{region '#Template'}
	{attribute 'Version' := '5.0.0.0'}
	{attribute 'Tags' := '"LCID": "1031", "Text": "RA, Sunprotection, Building"'}
	{attribute 'Tags' := '"LCID": "1033", "Text": "RA, Sunprotection, Building"'}
	{attribute 'Using' := '"Type": "Template", "URI": "Site"'}
	{attribute 'Using' := '"Type": "Template", "URI": "EC_ID"'}
	{attribute 'Using' := '"Type": "Template", "URI": "ST_BA_Sunblind"'}
	{attribute 'Description' := '"LCID": "1031", "Text": "Sonnenschutz Vereisungsschutz"'}
	{attribute 'Description' := '"LCID": "1033", "Text": "Sunprotection iceprotection"'}
{endregion}
FUNCTION_BLOCK FB_BA_IceProtection EXTENDS FB_BA_View
VAR_INPUT
END_VAR
VAR_OUTPUT
	stSunBld					: ST_BA_SunBld;
	bIcePrtcActv				: BOOL;	
END_VAR
VAR_INPUT CONSTANT	
	SpIce						: FB_BA_AV_Op;   
	DeiceTi						: FB_BA_AV_Op;		
	IceAlert					: FB_BA_BV;          
	SunBldIcePrtc				: FB_BA_SunBldIcePrtc;	
END_VAR	
VAR
	tonInitialWait				: TON;		
END_VAR

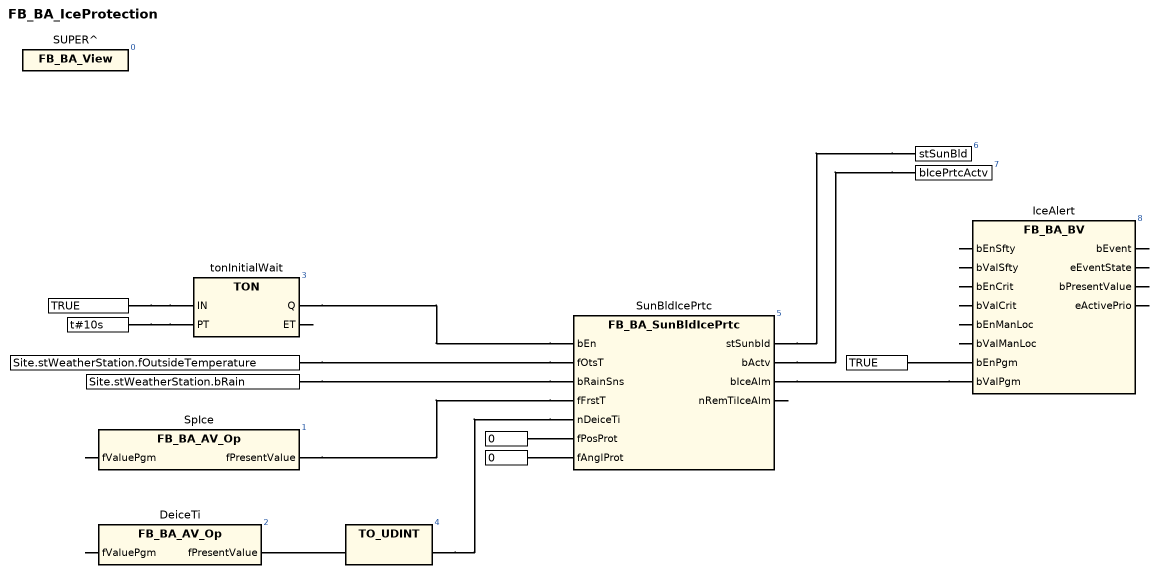
SUPER^(); // FB_BA_View
SpIce(); // FB_BA_AV_Op
DeiceTi(); // FB_BA_AV_Op
tonInitialWait(IN := TRUE, PT := t#10s); // TON
SunBldIcePrtc(
    bEn := tonInitialWait.Q,
    fOtsT := Site.stWeatherStation.fOutsideTemperature,
    bRainSns := Site.stWeatherStation.bRain,
    fFrstT := SpIce.fPresentValue,
    nDeiceTi := TO_UDINT(DeiceTi.fPresentValue),
    fPosProt := 0,
    fAnglProt := 0); // FB_BA_SunBldIcePrtc
stSunBld := SunBldIcePrtc.stSunbld;
bIcePrtcActv := SunBldIcePrtc.bActv;
IceAlert(bEnPgm := TRUE, bValPgm := SunBldIcePrtc.bIceAlm); // FB_BA_BV

METHOD FB_init : BOOL
VAR_INPUT
	bInitRetains : BOOL; // if TRUE, the retain variables are initialized (warm start / cold start)
	bInCopyCode : BOOL;  // if TRUE, the instance afterwards gets moved into the copy code (online change)
END_VAR
SpIce.iParent						:= THIS^; 
SpIce.iLabel						:= LblCtl_SetpointIce;
SpIce.eUnit							:= E_BA_Unit.eTemperature_DegreesCelsius; 
SpIce.fValueRm						:= -2.0;
                                	
DeiceTi.iParent						:= THIS^;
DeiceTi.iLabel						:= LblCtl_DeiceTime;
DeiceTi.eUnit						:= E_BA_Unit.eTime_Seconds; 
DeiceTi.fValueRm					:= 18000;

IceAlert.iParent					:= THIS^;
IceAlert.iLabel						:= LblCtl_IceAlert;
IceAlert.bEnOutOfService			:= FALSE;
IceAlert.sActiveText 				:= txtEvent_On;
IceAlert.sInactiveText 				:= txtEvent_Off;
IceAlert.bEnManualRm				:= FALSE;	//	Priority  8	
IceAlert.bValManualRm				:= FALSE;	//	Priority  8
IceAlert.nEventClassID				:= EC_ID.NC30;
IceAlert.stTimeDelay.nToNormal		:= BA2_Param.nDefTimeDelay_ToNormal;
IceAlert.stTimeDelay.nToAbnormal	:= BA2_Param.nDefTimeDelay_ToAbnormal;
IceAlert.bAlarmValue				:= TRUE;
IceAlert.bAcknowledgeRm				:= FALSE;		
IceAlert.aEventTransitionText[1]	:= txtEvent_On;  
IceAlert.aEventTransitionText[2]	:= txtEvent_None;
IceAlert.aEventTransitionText[3]	:= txtEvent_Off; 
IceAlert.eEnPlantLock				:= E_BA_LockPriority.eNoLock;
END_METHOD

END_FUNCTION_BLOCK

(* stored: Version 1.1.0.1, ProductVersion 3.1.4024.12
   POU FB_BA_IceProtection: Id {277f36d8-f0e7-4f5a-af62-055ab0d8b9c2}, SpecialFunc None
   Method FB_init: Id {9d40e247-68cf-404e-8ea4-d3429a37c723} *)
